PROGRAM MAIN
VAR
END_VAR

END_PROGRAM

(* stored: Version 1.1.0.1
   POU MAIN: Id {6d3b2b34-3b7b-4f9d-b63d-92fd87dfc156} *)
